PROGRAM FIFOaxis
VAR

	FifoOverride : FiFoSetChannelOverride;
	FifoDeIntegrate : FiFoGroupDisintegrate;
	FiFoReadDim1: FiFoGetDimension;
	FifoReadDimOK: BOOL;
	FifoNoOfAxis: UDINT;
	FifoNoOfEntries: UDINT;
	FIFOChInegrate : ARRAY[1..8] of FIFOIntegrate;
	FreeRows: DINT;
	NrOccupiedLines: DINT;
	n: UINT;
	StartIntegration: BOOL;

	FifoTableFromCNC	:	ARRAY[0..49,0..7] OF LREAL;
	FifoTableFromCNCLine:	ARRAY[0..400] OF LREAL;		//pos0 = number of rows
	FifoTableFromCNCTemp:	ARRAY[0..49,0..7] OF LREAL;
	FifoTable2	:	ARRAY[0..49,0..7] OF LREAL;

	FifoState: INT;
	StartFifo: BOOL;
	nOverride: UDINT;
	FrameNumber : UDINT;
	
	FifoWrite : FiFoWrite;
	FifoStart : FiFoStart;
	FifoStop : FifoStop;
	FifoTableCanTakeData : BOOL;
	FifoHasWritten : BOOL;
	
	m: INT;
	RowsFromCNC: UDINT;
	FiFoRunState: INT;
	p: INT;
	StartInt: INT;
	FifoActive: BOOL;
	fbMethods : FB_methods;
END_VAR


FifoStop(
	iChannelId:= 2, 
	bExecute:= , 
	tTimeout:= , 
	bBusy=> , 
	bErr=> , 
	iErrId=> );


CASE FifoState OF 
	
0:
	IF StartFifo THEN
		FrameNumber := 0;
		FifoState := 10;
	END_IF

10:
	StartIntegration := TRUE;
	StartFifo := FALSE;
	FifoOverride.bExecute := TRUE;
	FifoState := 20;

20: 
	StartIntegration := FALSE;
	FifoOverride.bExecute := FALSE;
	FiFoReadDim1.bExecute := TRUE;
	FifoState := 30;
	
30:
	FiFoReadDim1.bExecute := FALSE;
	FifoState := 40;
	
40:
	StartIntegration := TRUE;
	FifoState := 50;
	
50:
		FifoTableCanTakeData := TRUE;

		FIfostate := 100;

	
100:
	
	IF FifoHasWritten THEN
		FOR p := 0 TO LREAL_TO_INT(FifoTablefromCNCLine[0]) DO
			FifoTableFromCNCTemp[p, 0] := FifoTableFromCNCLine[8*p+1];
			FifoTableFromCNCTemp[p, 1] := FifoTableFromCNCLine[8*p+2];
			FifoTableFromCNCTemp[p, 2] := FifoTableFromCNCLine[8*p+3];
			FifoTableFromCNCTemp[p, 3] := FifoTableFromCNCLine[8*p+4];
			FifoTableFromCNCTemp[p, 4] := FifoTableFromCNCLine[8*p+5];
			FifoTableFromCNCTemp[p, 5] := FifoTableFromCNCLine[8*p+6];
			FifoTableFromCNCTemp[p, 6] := FifoTableFromCNCLine[8*p+7];
			FifoTableFromCNCTemp[p, 7] := FifoTableFromCNCLine[8*p+8];
			
		END_FOR
		
		FifoWrite.bExecute := TRUE;
		FifoState := 200;
		FifoHasWritten := FALSE;
		FifoTableCanTakeData := FALSE;
	END_IF
	
200:

	m := m +1;
	FifoWrite.bExecute := FALSE;
	FrameNumber := FrameNumber + 1;
	IF NOT fifostart.bBusy THEN
		//Fifostart.bExecute := TRUE;
		FifoState := 300;
	END_IF
	
300:
	//IF NrOccupiedLines > 0 THEN
		IF NOT fifostart.bBusy then // AND NOT fifostart.bErr THEN
			FifoStart.bExecute := FALSE;
			FifoTableCanTakeData := TRUE;
			Fifostate := 100;
		END_IF
	//END_IF
	
400:
//

500:
	
	//Sätt upp två minnen
	IF FifoTableFromCNC[0,0] <> 0 THEN
		MEMMOVE(ADR(FifoTable2), ADR(FifoTableFromCNC), SIZEOF(FifoTableFromCNC));	
		MEMSET(ADR(FifoTableFromCNC), 0, SIZEOF(FifoTableFromCNC));
	END_IF


END_CASE



CASE FiFoRunState OF

0: 
	IF 	NrOccupiedLines > 0 THEN
		FifoStart.bExecute := TRUE;
	ELSE
			FifoStart.bExecute := FALSE;	
	END_IF

END_CASE


//override
FifoOverride(
	iChannelId:= 2, 
	iOverride:= nOverride, 
	bExecute:= , 
	tTimeout:= T#1S, 
	bBusy=> , 
	bErr=> , 
	iErrId=> );
	
	
fbMethods();


//Integrate
CASE StartInt OF
	0:
	IF StartIntegration THEN
		FOR n:= 1 TO 8 DO
			FIFOChInegrate[n](ChNumber:=(n+9) , PosNumber := n,  bExcute:=TRUE );
		END_FOR
		StartInt := 10;
	END_IF

	10:
	StartIntegration := FALSE;	
	FOR n:= 1 TO 8 DO
		FIFOChInegrate[n](ChNumber:=(n+9) , PosNumber := n,  bExcute:=FALSE );
	END_FOR
	FifoActive := TRUE;
	StartInt := 0;
END_CASE


//Kolla lediga platser
		//läs parametrisering
		FiFoReadDim1(iChannelId:=2 );
		FifoReadDimOK := NOT FiFoReadDim1.bBusy AND NOT FiFoReadDim1.bErr;
		FiFoNoOfAxis := FiFoReadDim1.iNoOfAxes;
		FiFoNoOfEntries := FiFoReadDim1.iNoOfFifoEntries;
		NrOccupiedLines:= MAIN.motor_x_master.Axis.NcToPlc.SafEntries;
		IF FifoActive THEN
			FreeRows := FiFoNoOfEntries - NrOccupiedLines ;
		ELSE
			FreeRows := 0;	
		END_IF
		



//Deintegrate

FifoDeIntegrate(
	iChannelId:= 2, 
	bExecute:= , 
	tTimeout:= , 
	bBusy=> , 
	bErr=> , 
	iErrId=> );
	
	

IF FifoOverride.bExecute THEN
	FifoOverride.bExecute := FALSE;
END_IF

IF FifoDeIntegrate.bExecute THEN
	FifoActive := FALSE;
	FifoDeIntegrate.bExecute := FALSE;
END_IF

FifoWrite(
	iChannelId:= 2, 
	AdrDataArray:= ADR(FifoTableFromCNCTemp), 
	iColDim:= 8, 
	iRowsToWrite:= LREAL_TO_INT(FifoTablefromCNCLine[0]), 
	bExecute:= , 
	tTimeout:= , 
	bBusy=> , 
	bErr=> , 
	iErrId=> );
	
FifoStart(
	iChannelId:= 2, 
	bExecute:= , 
	tTimeout:= , 
	bBusy=> , 
	bErr=> , 
	iErrId=> );

METHOD M_Deintegrate : BOOL
VAR_INPUT
END_VAR
StartFifo := FALSE;
FifoState := 0;
FifoDeIntegrate.bExecute := TRUE;
END_METHOD

METHOD M_Integrate : BOOL
VAR_INPUT
END_VAR


StartIntegration := TRUE;
END_METHOD

END_PROGRAM

(* stored: Version 1.1.0.1, ProductVersion 3.1.4024.9
   POU FIFOaxis: Id {a14b88fd-3d7a-4a8f-bc03-9cc2654a729f}, SpecialFunc None
   Method M_Deintegrate: Id {c0a4e565-e833-415f-94be-a0d8c7212da5}
   Method M_Integrate: Id {71cc17b0-ced7-4d53-bc8d-c51290309d0c} *)
